FUNCTION_BLOCK TcoTixonBufferTask EXTENDS TcoTixonFeedingTask
VAR_IN_OUT
	inoConfig 	: TcoTixonGenericConfig;
   	inoControl 	: TcoTixonGenericControl;
	inoStatus 	: TcoTixonGenericStatus;	
END_VAR


IF Execute() THEN
	
	
    IF _progress = 0 THEN
        IF NOT __ISVALIDREF(inoControl) THEN
            _varInfo := __VARINFO(inoControl);
            Messenger.Programming(_sb.Clear().Append('<#Invalid reference: #>').Append(_varInfo.Symbol).ToString()).Pin();
        ELSIF NOT __ISVALIDREF(inoConfig) THEN
            _varInfo := __VARINFO(inoConfig);
            Messenger.Programming(_sb.Clear().Append('<#Invalid reference: #>').Append(_varInfo.Symbol).ToString()).Pin();
        ELSIF NOT __ISVALIDREF(inoStatus) THEN
            _varInfo := __VARINFO(inoStatus);
            Messenger.Programming(_sb.Clear().Append('<#Invalid reference: #>').Append(_varInfo.Symbol).ToString()).Pin();
        ELSIF NOT inoStatus.ControllerInAuto THEN
            _varInfo := __VARINFO(inoStatus.ControllerInAuto);
            Messenger.Warning(_sb.Clear().Append('<#Tixon control system not in auto #>').Append(_varInfo.Symbol).ToString());
        ELSE
			IF NOT THIS^._errorMessage.Pinned THEN	
           		_progress := _progress + 1;
			END_IF;

        END_IF

    END_IF
  	IF _progress = 1 THEN
        Messenger.Debug('<#Waiting for buffer is Empty #>');
        _timer(IN := NOT inoStatus.FillingSensor OR (inoStatus.SeparatorHomePos AND NOT inoStatus.SeparatorPresent),
            Pt := inoConfig.BufferEmptyTime);
			
        IF _timer.Q THEN
            _progress := _progress + 1;
            _timer(In := FALSE);
        END_IF;


    END_IF;
    IF _progress = 2 THEN
        Messenger.Debug('<#Waiting for blow on #>');
        _timer(IN :=TRUE,
            Pt := inoConfig.BufferBlowStartTime);
		  inoControl.BlowAValve := inoConfig.BufferBlowActive;	
        IF _timer.Q THEN  
			inoControl.FeedingA:=TRUE;
            _progress := _progress + 1;
            _timer(In := FALSE);
        END_IF;


    END_IF;
	

    IF _progress = 3 THEN
        Messenger.Debug('<#Waiting for buffer is full and go idle#>');
        _timer(IN := inoStatus.FillingSensor AND InoStatus.SeparatorPresent, Pt := inoConfig.BufferIdleTime);

        IF _timer.Q THEN
            _progress := _progress + 1;
            _timer(In := FALSE);
      // 	ELSIF inoStatus.SeparatorHomePos AND NOT inoStatus.SeparatorPresent THEN
//           _progress := 1;
        END_IF
    END_IF;

    IF _progress = 4 THEN
        inoControl.FeedingA := FALSE;
        Messenger.Debug('<#Waiting for buffer is full and blow ending#>');
        _timer(IN := inoStatus.FillingSensor, Pt := inoConfig.BufferBlowFullTime);
        IF _timer.Q THEN
            inoControl.BlowAValve := FALSE;
            _progress := _progress + 1;
            _timer(In := FALSE);
        END_IF;

    END_IF;

    IF _progress = 5 THEN
        THIS^.DoneWhen(TRUE);
    END_IF;

    CallTimers(_progress>1);//empty and strat feeding

    THIS^.ThrowWhen(_errorTimer.Q);

END_IF

IF THIS^.Error AND NOT _errorMessage.Pinned THEN
    THIS^.Restore();
END_IF

(*~
	<docu>
		<summary>
			Executes when task is aborted.
		</summary>			
	</docu>	
~*)
METHOD PROTECTED OnAbort
IF  __ISVALIDREF(inoStatus) THEN   THIS^.inoStatus.ActionDescription := '<#Buffer task  was aborted.#>'; END_IF;
END_METHOD

(*~
	<docu>
		<summary>
			Executes when task reaches the ```Done``` state .
		</summary>			
	</docu>	
~*)
METHOD PROTECTED OnDone
IF  __ISVALIDREF(inoStatus) THEN   THIS^.inoStatus.ActionDescription := '<#Buffer task  finished successfully.#>'; END_IF;
_progress:=0;
IF AutoRestore THEN
	Restore();
END_IF
END_METHOD

METHOD PROTECTED OnError
VAR
	description: STRING;
END_VAR
description := '<#Buffer task finished with error.#>'; 
inoControl.FeedingA:=FALSE;
inoControl.BlowAValve:=false;
IF  __ISVALIDREF(inoStatus) THEN   THIS^.inoStatus.ActionDescription := description; END_IF;
THIS^._errorMessage.Error(_sb.Clear().Append(description).Append(' To restore acknowledge this alarm.').ToString()).Pin();
END_METHOD

METHOD PROTECTED OnStart
IF  __ISVALIDREF(inoStatus) THEN  THIS^.inoStatus.ActionDescription := '<#Buffer task started.#>'; END_IF; 

CallTimers(FALSE);
END_METHOD

(*~
	<docu>
		<summary>
			Restores this instance to the Ready state. Can be called explicitly or from within one of the restore mechanisms.
			<para>
				See also <see cref="PlcDocu.TcoCore.TcoTask.AutoRestorable()"/>
			</para>
		</summary>			
	</docu>	
~*)
METHOD Restore : ITcoRestorable
SUPER^.Restore();
END_METHOD

END_FUNCTION_BLOCK

(* stored: Version 1.1.0.1, ProductVersion 3.1.4024.12
   POU TcoTixonBufferTask: Id {69195fb9-0897-0eaa-2196-479e953ed90b}, SpecialFunc None
   Method OnAbort: Id {6a0aa103-225a-0ff0-1024-f705a6d94be6}
   Method OnDone: Id {241df0b7-81f4-02a7-1f5b-9ab4f64f9c40}
   Method OnError: Id {7865d813-1fc4-0e6c-15be-224cad6b43cd}
   Method OnStart: Id {1eebfa18-4075-0668-0834-5bb75b3bb329}
   Method Restore: Id {1f561e44-1a7f-010c-22e6-694cb34d2ae8} *)
